// TIA Portal V17 export
// export: Created 2026-04-13T11:12:54.6885374Z, ExportSetting WithDefaults, DisplayName Totally Integrated Automation Portal, DisplayVersion V17 Update 4, DisplayName TIA Portal Openness, DisplayVersion V17 Update 4, DisplayName TIA Portal Version Control Interface, DisplayVersion V17, DisplayName SINAMICS Startdrive Advanced, DisplayVersion V17, DisplayName SINAMICS Startdrive G130, G150, S120, S150, SINAMICS MV, S210, DisplayVersion V17, DisplayName SINAMICS Startdrive G110M, G120, G120C, G120D, G120P, G115D, DisplayVersion V17, DisplayName STEP 7 Professional, DisplayVersion V17 Update 4, DisplayName STEP 7 Safety, DisplayVersion V17, DisplayName WinCC Professional, DisplayVersion V17 Update 4
VBScript "ReadFile_Audit"  Type=Sub
  Dim Path
  Dim fs,f
  Dim  i, j, field2,ss
  Dim field'(99999)
  Dim MaxLines
  Dim HiField(10,8)
  Dim Lines,sumPag,CurtPag,startLines,endLines
  Dim SizeOfFile
  
  '指定日志文件所在目录\Storage Card USB\
  Path ="\Storage Card USB\AuditTrail\AuditTrail0.txt" '"\\DESKTOP-CEFLV5H\winccprojects\AuditTrail0.csv"
  '读取日志文件
  SmartTags("执行说明")="读取日志文件中"
  'Set fs = CreateObject("Scripting.FileSystemObject")'FileCtl.FileSystem
  Set fs = CreateObject("FileCtl.file")
  SmartTags("执行说明")="已创建对象"
  'Set f = fs.OpenTextFile(Path,1,1)
  fs.open Path,1,1
  SizeOfFile = fs.LOF
  
  SmartTags("执行说明")="已打开文件"
  'field = f.ReadAll
  'field = Split(field,vbCrLf)
  MaxLines = 0
  Do While fs.EOF <>True
  	'field(MaxLines) = fs.lineinputstring
  	'MaxLines = MaxLines +1
  	field = CStr(fs.inputB(SizeOfFile))
  Loop
  field = Split(field,vbCrLf)
  '获取日志文件数量
  SmartTags("执行说明")="日志文件读取完成"
  Lines=UBound(field,1)-2'MaxLines - 2
  '获取总页数
  If Lines <1 Then
  	SmartTags("执行说明")="不存在日志信息"
  	Exit Sub
  End If
   sumPag= Lines \ 15
  
  If (sumPag*15) < Lines Then
  	sumPag=sumPag+1
  End If
  SmartTags("日志总页数")=sumPag
  
  
  '显示日志数据
  	CurtPag = SmartTags("日志当前页数")
  	If (CurtPag > sumPag) Or (CurtPag < 1)  Then
  
  		CurtPag = 1
  		SmartTags("日志当前页数")=1
  	End If
  
  	startLines = (CurtPag -1) * 15
  	SmartTags("执行说明")="日志显示" & startLines & field(0)
  	For i = 1 To 15
  
  		If (i+startLines) <= Lines Then
  			field2 =Split( field(i + startLines ),vbtab)
  			SmartTags("Audit_编号" & i )=field2(0)
  			SmartTags("Audit_时间" & i )=field2(1)
  			SmartTags("Audit_用户" & i )=field2(3)
  			SmartTags("Audit_对象" & i )=field2(4)
  			SmartTags("Audit_描述" & i )=field2(5)
  		Else
  			SmartTags("Audit_编号" & i )=""
  			SmartTags("Audit_时间" & i )=""
  			SmartTags("Audit_用户" & i )=""
  			SmartTags("Audit_对象" & i )=""
  			SmartTags("Audit_描述" & i )=""
  		End If
  
  	Next
  	SmartTags("执行说明")="日志加载完成"
  	f.Close
  	Set  f  = Nothing
